{attribute 'GeneratedUsingTerminal: APS1003-7000-0016'}
{attribute addProperty BoxType "APS1003-7000-0016"}
{attribute addProperty Id "YVR_InputsAT %I*YVR_Inputs_4719D0DB98YVR_OutputsAT %Q*YVR_Outputs_31F2CBB3146WcStateAT %I*WcState_9091E0EB2InfoDataAT %I*InfoData_1088C70510"}
{attribute addProperty CRC "1334787595"}
{attribute addProperty Size "256"}
TYPE APS1003_4F8F3E0B EXTENDS EtcSlaveTerminalBase_947E5A46 :
STRUCT
	{attribute addProperty Name "YVR_Inputs"}
	YVR_Inputs : YVR_Inputs_4719D0DB;
	{attribute addProperty Name "YVR_Outputs"}
	YVR_Outputs : YVR_Outputs_31F2CBB3;
	{attribute addProperty Name "WcState"}
	WcState : WcState_9091E0EB;
	{attribute addProperty Name "InfoData"}
	InfoData : InfoData_1088C705;
END_STRUCT
END_TYPE

(* stored: Version 1.2.0.0, ProductVersion 3.1.4024.9
   DUT APS1003_4F8F3E0B: Id {96236861-ad80-46eb-9135-e370a3ca3e4c} *)
